{attribute addProperty BoxType "EL1202-0100-0016"}
{attribute addProperty Id "NextLatchTimeAT %I*ULINT648"}
{attribute addProperty CRC "1092592461"}
{attribute addProperty SizeInBites "64"}
{attribute addProperty SizeInBytes "8"}
TYPE DC_411FA34D :
STRUCT
	{attribute addProperty Name "NextLatchTime"}
	NextLatchTime AT %I* : ULINT;
END_STRUCT
END_TYPE

(* stored: Version 1.2.0.0, ProductVersion 3.1.4024.9
   DUT DC_411FA34D: Id {3b4a1063-a5df-40ad-acde-d0019daaf43f} *)
